PROGRAM MAIN
VAR
END_VAR

//TcUnit.RUN();

END_PROGRAM

(* stored: Version 1.1.0.1, ProductVersion 3.1.4024.12
   POU MAIN: Id {0308f13d-366d-4f3c-948a-90028615a6c6}, SpecialFunc None *)
